TYPE Struct_PLCVersion :
STRUCT
	Servo_Compatibility_high						:	SINT := 0;
	Servo_Compatibility_low							:	SINT := 5;
	PLC_Function									:	SINT := 0;
	LIB_Version										:	ARRAY[0..2] OF BYTE;
END_STRUCT
END_TYPE

(* stored: Version 1.1.0.1, ProductVersion 3.1.4020.12
   DUT Struct_PLCVersion: Id {d78ff7d8-3a50-4e8d-96f9-cb9b93c2f057} *)
